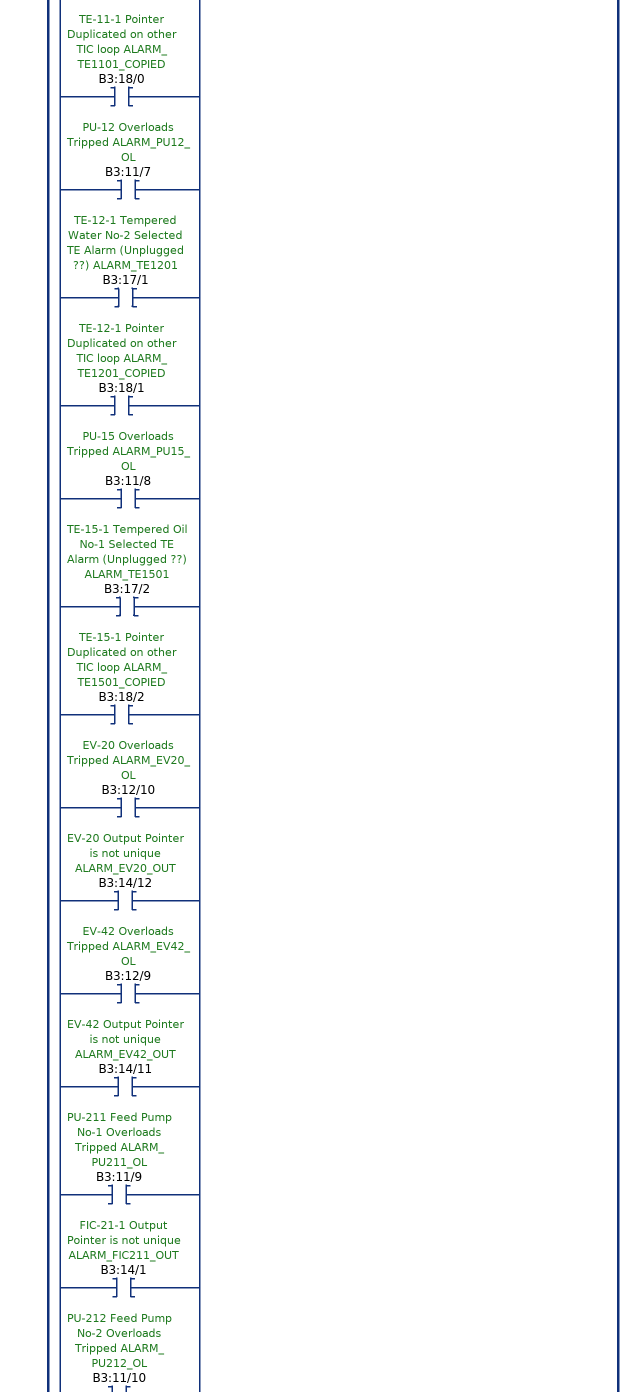

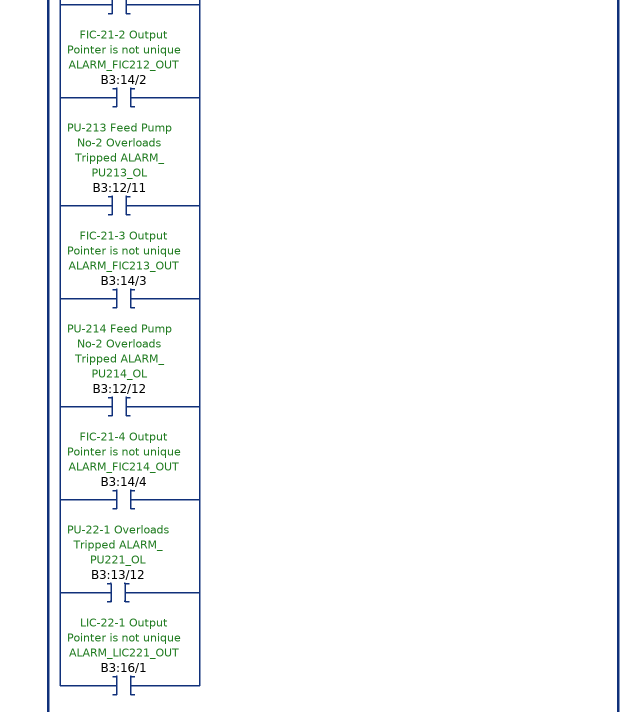
% Rung: 4 %
% This Rung Sets a Bit
% used by the HMI's
% to Determine Whether Alarm Status Page 1
% Has an Active Alarm %
SOR BST XIC B3:12/3 NXB XIC B3:12/0 NXB XIC B3:11/3 NXB XIC B3:14/10 NXB XIC B3:13/13 NXB XIC B3:13/14 NXB XIC B3:11/0 NXB XIC B3:11/1 NXB XIC B3:14/8 NXB XIC B3:11/2 NXB XIC B3:14/9 NXB XIC B3:11/6 NXB XIC B3:17/0 NXB XIC B3:18/0 NXB XIC B3:11/7 NXB XIC B3:17/1 NXB XIC B3:18/1 NXB XIC B3:11/8 NXB XIC B3:17/2 NXB XIC B3:18/2 NXB XIC B3:12/10 NXB XIC B3:14/12 NXB XIC B3:12/9 NXB XIC B3:14/11 NXB XIC B3:11/9 NXB XIC B3:14/1 NXB XIC B3:11/10 NXB XIC B3:14/2 NXB XIC B3:12/11 NXB XIC B3:14/3 NXB XIC B3:12/12 NXB XIC B3:14/4 NXB XIC B3:13/12 NXB XIC B3:16/1 BND OTE B3:10/11 EOR
%   B3:12/3  ALARM_FIRE_ALARM  "WFE Test Center Fire Alarm has be Triggered" %
%   B3:12/0  ALARM_E_STOP  "E-Stop Pushbutton has Been Pressed" %
%   B3:11/3  ALARM_AG04_OL  "AG-4 Overloads Tripped" %
%   B3:14/10  ALARM_AG04_OUT  "AG-4 Output Pointer is not unique" %
%   B3:13/13  ALARM_EF1_OL  "EF-1 Process Area Exhaust Fan Overloads Tripped" %
%   B3:13/14  ALARM_EF2_OL  "EF-2 Utility Room Exhaust Fan Overloads Tripped" %
%   B3:11/0  ALARM_EV01_OL  "EV-1 Overloads Tripped" %
%   B3:11/1  ALARM_EV02_OL  "EV-2 Overloads Tripped" %
%   B3:14/8  ALARM_EV02_OUT  "EV-2 Output Pointer is not unique" %
%   B3:11/2  ALARM_EV03_OL  "EV-3 Overloads Tripped" %
%   B3:14/9  ALARM_EV03_OUT  "EV-3 Output Pointer is not unique" %
%   B3:11/6  ALARM_PU11_OL  "PU-11 Overloads Tripped" %
%   B3:17/0  ALARM_TE1101  "TE-11-1 Tempered Water No-1 Selected TE Alarm (Unplugged ??)" %
%   B3:18/0  ALARM_TE1101_COPIED  "TE-11-1 Pointer Duplicated on other TIC loop" %
%   B3:11/7  ALARM_PU12_OL  "PU-12 Overloads Tripped" %
%   B3:17/1  ALARM_TE1201  "TE-12-1 Tempered Water No-2 Selected TE Alarm (Unplugged ??)" %
%   B3:18/1  ALARM_TE1201_COPIED  "TE-12-1 Pointer Duplicated on other TIC loop" %
%   B3:11/8  ALARM_PU15_OL  "PU-15 Overloads Tripped" %
%   B3:17/2  ALARM_TE1501  "TE-15-1 Tempered Oil No-1 Selected TE Alarm (Unplugged ??)" %
%   B3:18/2  ALARM_TE1501_COPIED  "TE-15-1 Pointer Duplicated on other TIC loop" %
%   B3:12/10  ALARM_EV20_OL  "EV-20 Overloads Tripped" %
%   B3:14/12  ALARM_EV20_OUT  "EV-20 Output Pointer is not unique" %
%   B3:12/9  ALARM_EV42_OL  "EV-42 Overloads Tripped" %
%   B3:14/11  ALARM_EV42_OUT  "EV-42 Output Pointer is not unique" %
%   B3:11/9  ALARM_PU211_OL  "PU-211 Feed Pump No-1 Overloads Tripped" %
%   B3:14/1  ALARM_FIC211_OUT  "FIC-21-1 Output Pointer is not unique" %
%   B3:11/10  ALARM_PU212_OL  "PU-212 Feed Pump No-2 Overloads Tripped" %
%   B3:14/2  ALARM_FIC212_OUT  "FIC-21-2 Output Pointer is not unique" %
%   B3:12/11  ALARM_PU213_OL  "PU-213 Feed Pump No-2 Overloads Tripped" %
%   B3:14/3  ALARM_FIC213_OUT  "FIC-21-3 Output Pointer is not unique" %
%   B3:12/12  ALARM_PU214_OL  "PU-214 Feed Pump No-2 Overloads Tripped" %
%   B3:14/4  ALARM_FIC214_OUT  "FIC-21-4 Output Pointer is not unique" %
%   B3:13/12  ALARM_PU221_OL  "PU-22-1 Overloads Tripped" %
%   B3:16/1  ALARM_LIC221_OUT  "LIC-22-1 Output Pointer is not unique" %
%   B3:10/11  ALARM_ACTIVE_PAGE1  "Alarm Active on HMI Page 1 of 3" %

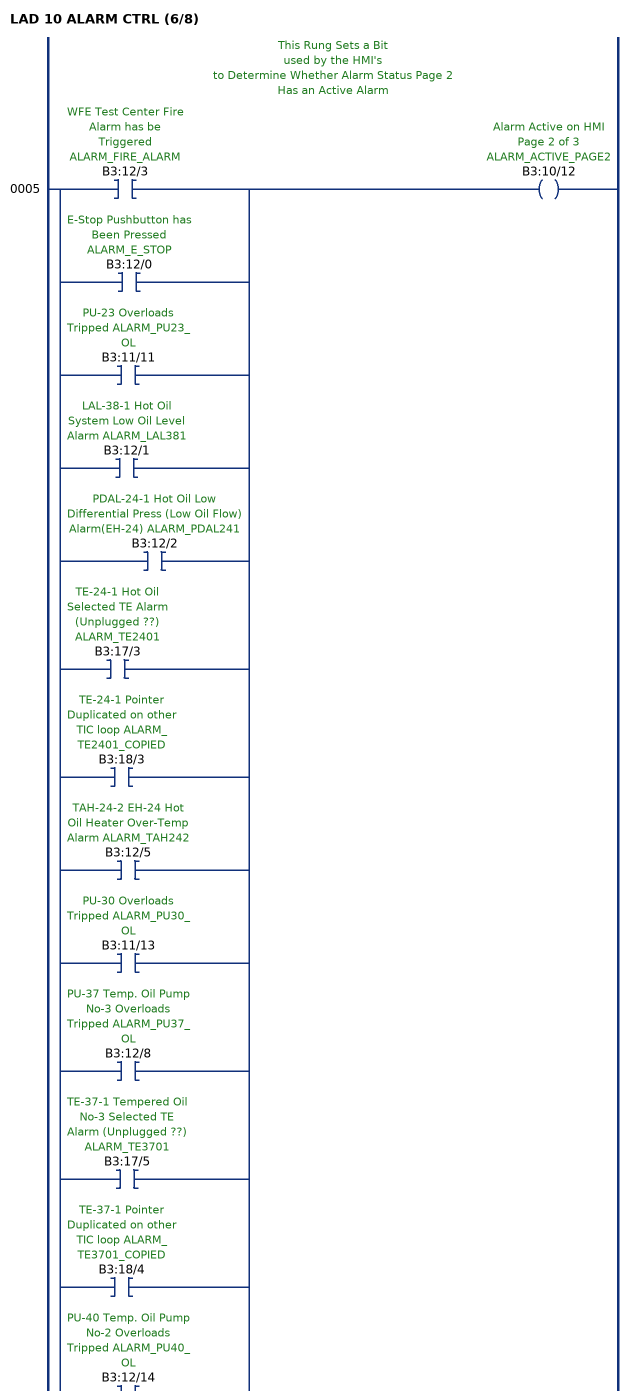

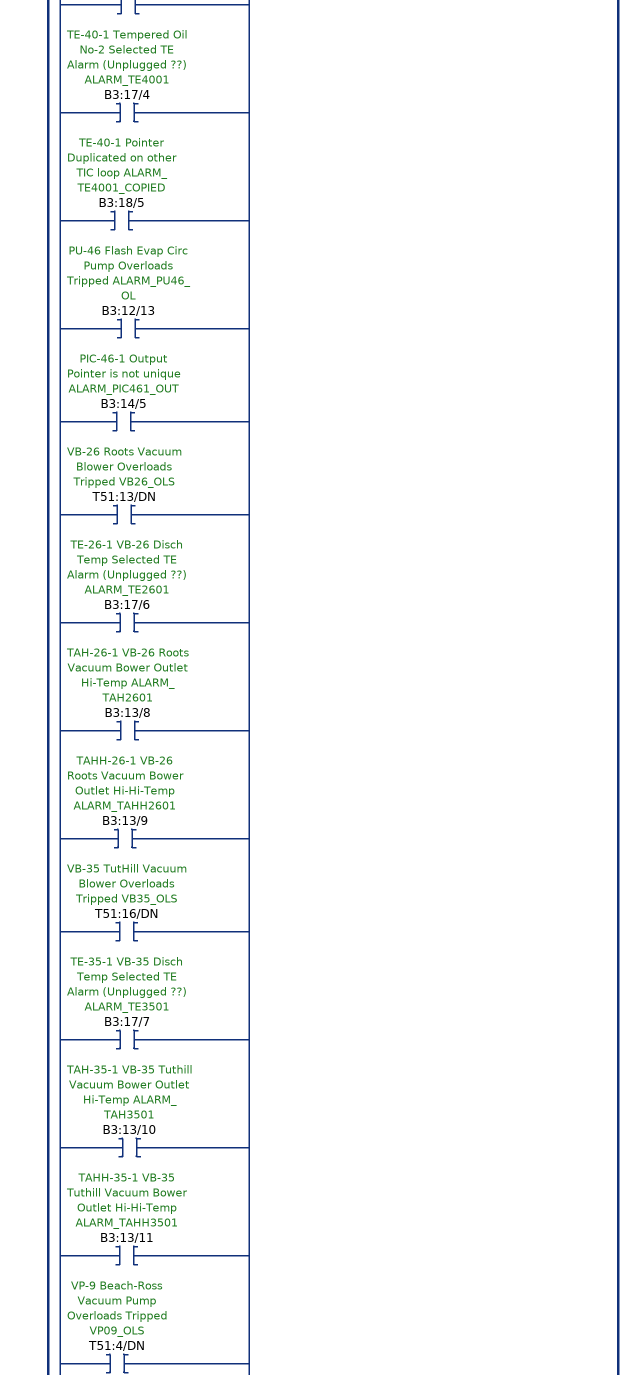

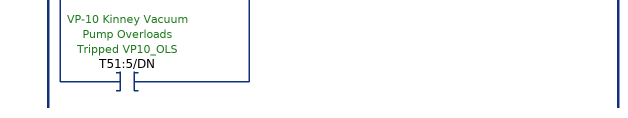
% Rung: 5 %
% This Rung Sets a Bit
% used by the HMI's
% to Determine Whether Alarm Status Page 2
% Has an Active Alarm %
SOR BST XIC B3:12/3 NXB XIC B3:12/0 NXB XIC B3:11/11 NXB XIC B3:12/1 NXB XIC B3:12/2 NXB XIC B3:17/3 NXB XIC B3:18/3 NXB XIC B3:12/5 NXB XIC B3:11/13 NXB XIC B3:12/8 NXB XIC B3:17/5 NXB XIC B3:18/4 NXB XIC B3:12/14 NXB XIC B3:17/4 NXB XIC B3:18/5 NXB XIC B3:12/13 NXB XIC B3:14/5 NXB XIC T51:13/DN NXB XIC B3:17/6 NXB XIC B3:13/8 NXB XIC B3:13/9 NXB XIC T51:16/DN NXB XIC B3:17/7 NXB XIC B3:13/10 NXB XIC B3:13/11 NXB XIC T51:4/DN NXB XIC T51:5/DN BND OTE B3:10/12 EOR
%   B3:12/3  ALARM_FIRE_ALARM  "WFE Test Center Fire Alarm has be Triggered" %
%   B3:12/0  ALARM_E_STOP  "E-Stop Pushbutton has Been Pressed" %
%   B3:11/11  ALARM_PU23_OL  "PU-23 Overloads Tripped" %
%   B3:12/1  ALARM_LAL381  "LAL-38-1 Hot Oil System Low Oil Level Alarm" %
%   B3:12/2  ALARM_PDAL241  "PDAL-24-1 Hot Oil Low Differential Press (Low Oil Flow) Alarm(EH-24)" %
%   B3:17/3  ALARM_TE2401  "TE-24-1 Hot Oil Selected TE Alarm (Unplugged ??)" %
%   B3:18/3  ALARM_TE2401_COPIED  "TE-24-1 Pointer Duplicated on other TIC loop" %
%   B3:12/5  ALARM_TAH242  "TAH-24-2 EH-24 Hot Oil Heater Over-Temp Alarm" %
%   B3:11/13  ALARM_PU30_OL  "PU-30 Overloads Tripped" %
%   B3:12/8  ALARM_PU37_OL  "PU-37 Temp. Oil Pump No-3 Overloads Tripped" %
%   B3:17/5  ALARM_TE3701  "TE-37-1 Tempered Oil No-3 Selected TE Alarm (Unplugged ??)" %
%   B3:18/4  ALARM_TE3701_COPIED  "TE-37-1 Pointer Duplicated on other TIC loop" %
%   B3:12/14  ALARM_PU40_OL  "PU-40 Temp. Oil Pump No-2 Overloads Tripped" %
%   B3:17/4  ALARM_TE4001  "TE-40-1 Tempered Oil No-2 Selected TE Alarm (Unplugged ??)" %
%   B3:18/5  ALARM_TE4001_COPIED  "TE-40-1 Pointer Duplicated on other TIC loop" %
%   B3:12/13  ALARM_PU46_OL  "PU-46 Flash Evap Circ Pump Overloads Tripped" %
%   B3:14/5  ALARM_PIC461_OUT  "PIC-46-1 Output Pointer is not unique" %
%   T51:13/DN  VB26_OLS  "VB-26 Roots Vacuum Blower Overloads Tripped" %
%   B3:17/6  ALARM_TE2601  "TE-26-1 VB-26 Disch Temp Selected TE Alarm (Unplugged ??)" %
%   B3:13/8  ALARM_TAH2601  "TAH-26-1 VB-26 Roots Vacuum Bower Outlet Hi-Temp" %
%   B3:13/9  ALARM_TAHH2601  "TAHH-26-1 VB-26 Roots Vacuum Bower Outlet Hi-Hi-Temp" %
%   T51:16/DN  VB35_OLS  "VB-35 TutHill Vacuum Blower Overloads Tripped" %
%   B3:17/7  ALARM_TE3501  "TE-35-1 VB-35 Disch Temp Selected TE Alarm (Unplugged ??)" %
%   B3:13/10  ALARM_TAH3501  "TAH-35-1 VB-35 Tuthill Vacuum Bower Outlet Hi-Temp" %
%   B3:13/11  ALARM_TAHH3501  "TAHH-35-1 VB-35 Tuthill Vacuum Bower Outlet Hi-Hi-Temp" %
%   T51:4/DN  VP09_OLS  "VP-9 Beach-Ross Vacuum Pump Overloads Tripped" %
%   T51:5/DN  VP10_OLS  "VP-10 Kinney Vacuum Pump Overloads Tripped" %
%   B3:10/12  ALARM_ACTIVE_PAGE2  "Alarm Active on HMI Page 2 of 3" %

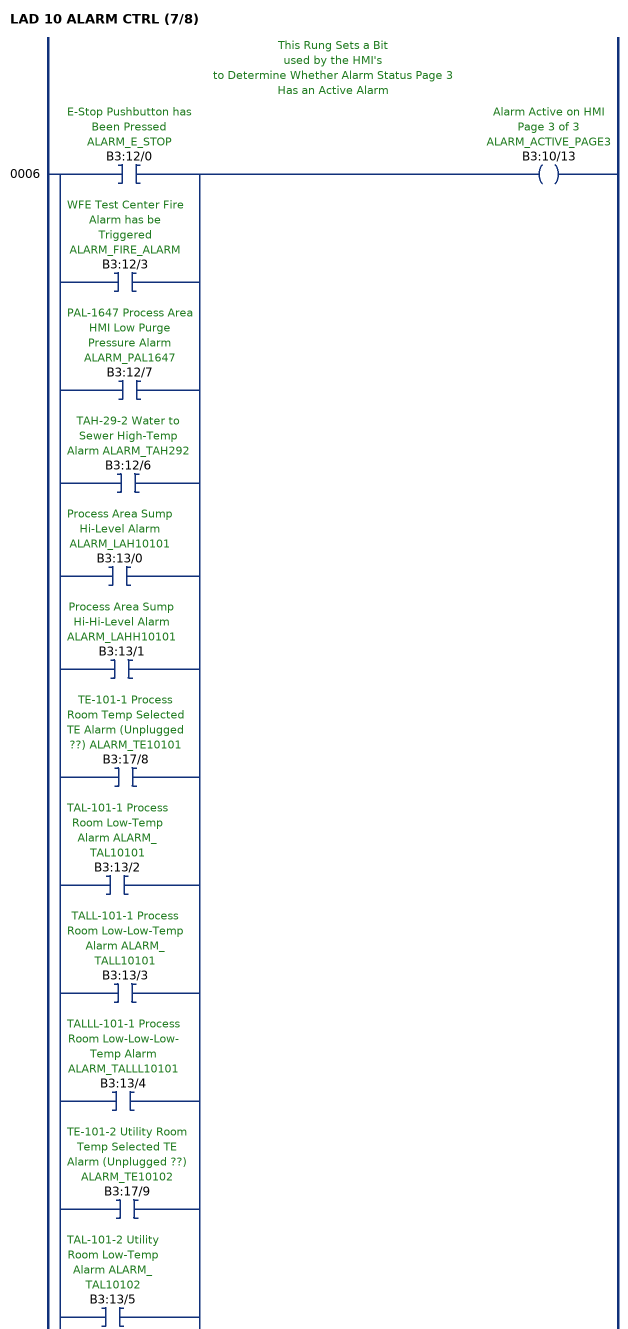

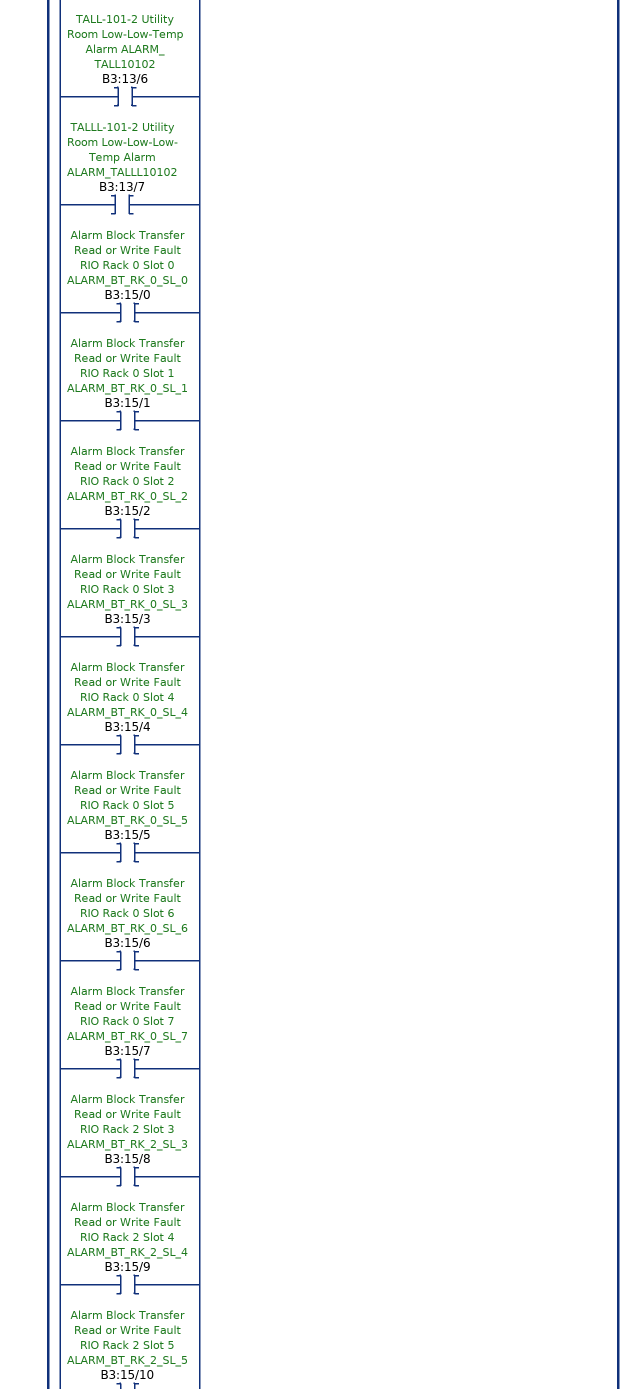

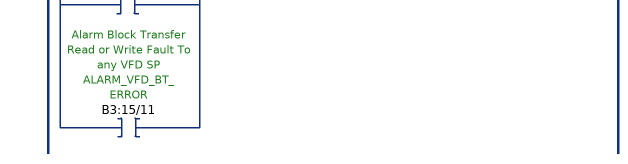
% Rung: 6 %
% This Rung Sets a Bit
% used by the HMI's
% to Determine Whether Alarm Status Page 3
% Has an Active Alarm %
SOR BST XIC B3:12/0 NXB XIC B3:12/3 NXB XIC B3:12/7 NXB XIC B3:12/6 NXB XIC B3:13/0 NXB XIC B3:13/1 NXB XIC B3:17/8 NXB XIC B3:13/2 NXB XIC B3:13/3 NXB XIC B3:13/4 NXB XIC B3:17/9 NXB XIC B3:13/5 NXB XIC B3:13/6 NXB XIC B3:13/7 NXB XIC B3:15/0 NXB XIC B3:15/1 NXB XIC B3:15/2 NXB XIC B3:15/3 NXB XIC B3:15/4 NXB XIC B3:15/5 NXB XIC B3:15/6 NXB XIC B3:15/7 NXB XIC B3:15/8 NXB XIC B3:15/9 NXB XIC B3:15/10 NXB XIC B3:15/11 BND OTE B3:10/13 EOR
%   B3:12/0  ALARM_E_STOP  "E-Stop Pushbutton has Been Pressed" %
%   B3:12/3  ALARM_FIRE_ALARM  "WFE Test Center Fire Alarm has be Triggered" %
%   B3:12/7  ALARM_PAL1647  "PAL-1647 Process Area HMI Low Purge Pressure Alarm" %
%   B3:12/6  ALARM_TAH292  "TAH-29-2 Water to Sewer High-Temp Alarm" %
%   B3:13/0  ALARM_LAH10101  "Process Area Sump Hi-Level Alarm" %
%   B3:13/1  ALARM_LAHH10101  "Process Area Sump Hi-Hi-Level Alarm" %
%   B3:17/8  ALARM_TE10101  "TE-101-1 Process Room Temp Selected TE Alarm (Unplugged ??)" %
%   B3:13/2  ALARM_TAL10101  "TAL-101-1 Process Room Low-Temp Alarm" %
%   B3:13/3  ALARM_TALL10101  "TALL-101-1 Process Room Low-Low-Temp Alarm" %
%   B3:13/4  ALARM_TALLL10101  "TALLL-101-1 Process Room Low-Low-Low-Temp Alarm" %
%   B3:17/9  ALARM_TE10102  "TE-101-2 Utility Room Temp Selected TE Alarm (Unplugged ??)" %
%   B3:13/5  ALARM_TAL10102  "TAL-101-2 Utility Room Low-Temp Alarm" %
%   B3:13/6  ALARM_TALL10102  "TALL-101-2 Utility Room Low-Low-Temp Alarm" %
%   B3:13/7  ALARM_TALLL10102  "TALLL-101-2 Utility Room Low-Low-Low-Temp Alarm" %
%   B3:15/0  ALARM_BT_RK_0_SL_0  "Alarm Block Transfer Read or Write Fault RIO Rack 0 Slot 0" %
%   B3:15/1  ALARM_BT_RK_0_SL_1  "Alarm Block Transfer Read or Write Fault RIO Rack 0 Slot 1" %
%   B3:15/2  ALARM_BT_RK_0_SL_2  "Alarm Block Transfer Read or Write Fault RIO Rack 0 Slot 2" %
%   B3:15/3  ALARM_BT_RK_0_SL_3  "Alarm Block Transfer Read or Write Fault RIO Rack 0 Slot 3" %
%   B3:15/4  ALARM_BT_RK_0_SL_4  "Alarm Block Transfer Read or Write Fault RIO Rack 0 Slot 4" %
%   B3:15/5  ALARM_BT_RK_0_SL_5  "Alarm Block Transfer Read or Write Fault RIO Rack 0 Slot 5" %
%   B3:15/6  ALARM_BT_RK_0_SL_6  "Alarm Block Transfer Read or Write Fault RIO Rack 0 Slot 6" %
%   B3:15/7  ALARM_BT_RK_0_SL_7  "Alarm Block Transfer Read or Write Fault RIO Rack 0 Slot 7" %
%   B3:15/8  ALARM_BT_RK_2_SL_3  "Alarm Block Transfer Read or Write Fault RIO Rack 2 Slot 3" %
%   B3:15/9  ALARM_BT_RK_2_SL_4  "Alarm Block Transfer Read or Write Fault RIO Rack 2 Slot 4" %
%   B3:15/10  ALARM_BT_RK_2_SL_5  "Alarm Block Transfer Read or Write Fault RIO Rack 2 Slot 5" %
%   B3:15/11  ALARM_VFD_BT_ERROR  "Alarm Block Transfer Read or Write Fault To any VFD SP" %
%   B3:10/13  ALARM_ACTIVE_PAGE3  "Alarm Active on HMI Page 3 of 3" %

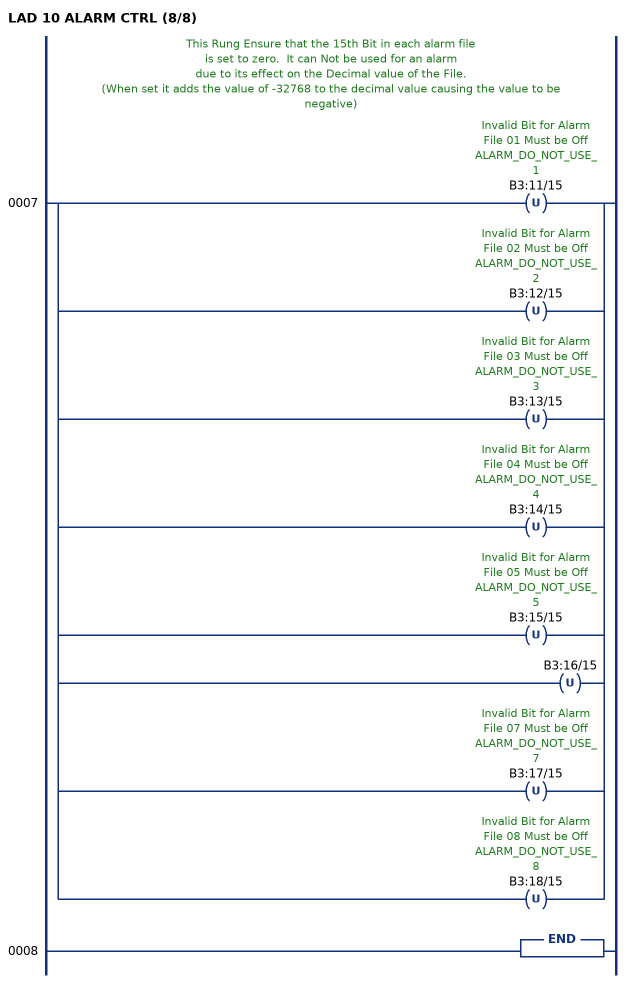
% Rung: 7 %
% This Rung Ensure that the 15th Bit in each alarm file
% is set to zero.  It can Not be used for an alarm
% due to its effect on the Decimal value of the File.
% (When set it adds the value of -32768 to the decimal value causing the value to be negative) %
SOR BST OTU B3:11/15 NXB OTU B3:12/15 NXB OTU B3:13/15 NXB OTU B3:14/15 NXB OTU B3:15/15 NXB OTU B3:16/15 NXB OTU B3:17/15 NXB OTU B3:18/15 BND EOR
%   B3:11/15  ALARM_DO_NOT_USE_1  "Invalid Bit for Alarm File 01 Must be Off" %
%   B3:12/15  ALARM_DO_NOT_USE_2  "Invalid Bit for Alarm File 02 Must be Off" %
%   B3:13/15  ALARM_DO_NOT_USE_3  "Invalid Bit for Alarm File 03 Must be Off" %
%   B3:14/15  ALARM_DO_NOT_USE_4  "Invalid Bit for Alarm File 04 Must be Off" %
%   B3:15/15  ALARM_DO_NOT_USE_5  "Invalid Bit for Alarm File 05 Must be Off" %
%   B3:17/15  ALARM_DO_NOT_USE_7  "Invalid Bit for Alarm File 07 Must be Off" %
%   B3:18/15  ALARM_DO_NOT_USE_8  "Invalid Bit for Alarm File 08 Must be Off" %
% Rung: 8 %
SOR END EOR

LADDER 11 "ALARMS"    % Process Alarms %
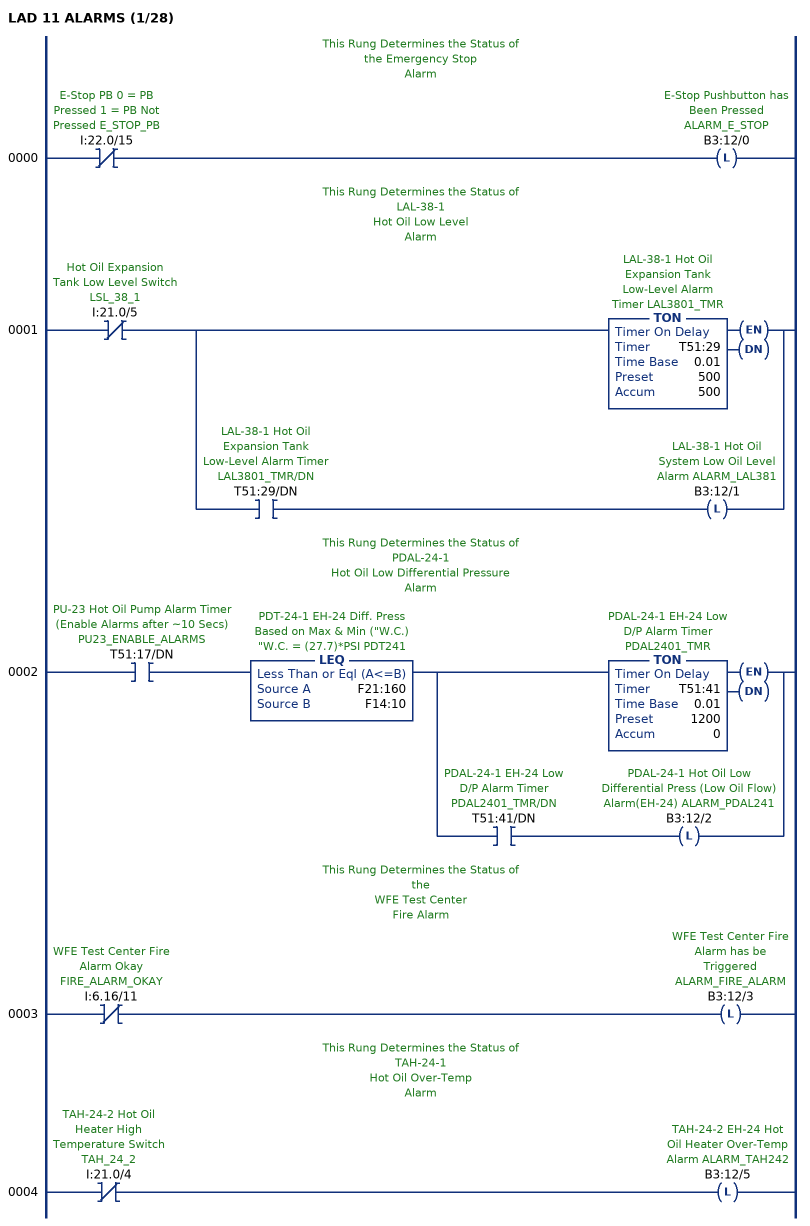
% Rung: 0 %
% This Rung Determines the Status of
% the Emergency Stop
% Alarm %
SOR XIO I:22.0/15 OTL B3:12/0 EOR
%   I:22.0/15  E_STOP_PB  "E-Stop PB 0 = PB Pressed 1 = PB Not Pressed" %
%   B3:12/0  ALARM_E_STOP  "E-Stop Pushbutton has Been Pressed" %
% Rung: 1 %
% This Rung Determines the Status of
% LAL-38-1
% Hot Oil Low Level
% Alarm %
SOR XIO I:21.0/5 BST TON T51:29 0.01 500 500 NXB XIC T51:29/DN OTL B3:12/1 BND EOR
%   I:21.0/5  LSL_38_1  "Hot Oil Expansion Tank Low Level Switch" %
%   T51:29  LAL3801_TMR  "LAL-38-1 Hot Oil Expansion Tank Low-Level Alarm Timer" %
%   B3:12/1  ALARM_LAL381  "LAL-38-1 Hot Oil System Low Oil Level Alarm" %
% Rung: 2 %
% This Rung Determines the Status of
% PDAL-24-1
% Hot Oil Low Differential Pressure
% Alarm %
SOR XIC T51:17/DN LEQ F21:160 F14:10 BST TON T51:41 0.01 1200 0 NXB XIC T51:41/DN OTL B3:12/2 BND EOR
%   T51:17/DN  PU23_ENABLE_ALARMS  "PU-23 Hot Oil Pump Alarm Timer (Enable Alarms after ~10 Secs)" %
%   F21:160  PDT241  "PDT-24-1 EH-24 Diff. Press Based on Max & Min ("W.C.) "W.C. = (27.7)*PSI" %
%   F14:10  PDAL2401_SP  "PDAL-24-1 Hot Oil Low Differential Press (Low Oil Flow) SP" %
%   T51:41  PDAL2401_TMR  "PDAL-24-1 EH-24 Low D/P Alarm Timer" %
%   B3:12/2  ALARM_PDAL241  "PDAL-24-1 Hot Oil Low Differential Press (Low Oil Flow) Alarm(EH-24)" %
% Rung: 3 %
% This Rung Determines the Status of
% the
% WFE Test Center
% Fire Alarm %
SOR XIO I:6.16/11 OTL B3:12/3 EOR
%   I:6.16/11  FIRE_ALARM_OKAY  "WFE Test Center Fire Alarm Okay" %
%   B3:12/3  ALARM_FIRE_ALARM  "WFE Test Center Fire Alarm has be Triggered" %
% Rung: 4 %
% This Rung Determines the Status of
% TAH-24-1
% Hot Oil Over-Temp
% Alarm %
SOR XIO I:21.0/4 OTL B3:12/5 EOR
%   I:21.0/4  TAH_24_2  "TAH-24-2 Hot Oil Heater High Temperature Switch" %
%   B3:12/5  ALARM_TAH242  "TAH-24-2 EH-24 Hot Oil Heater Over-Temp Alarm" %

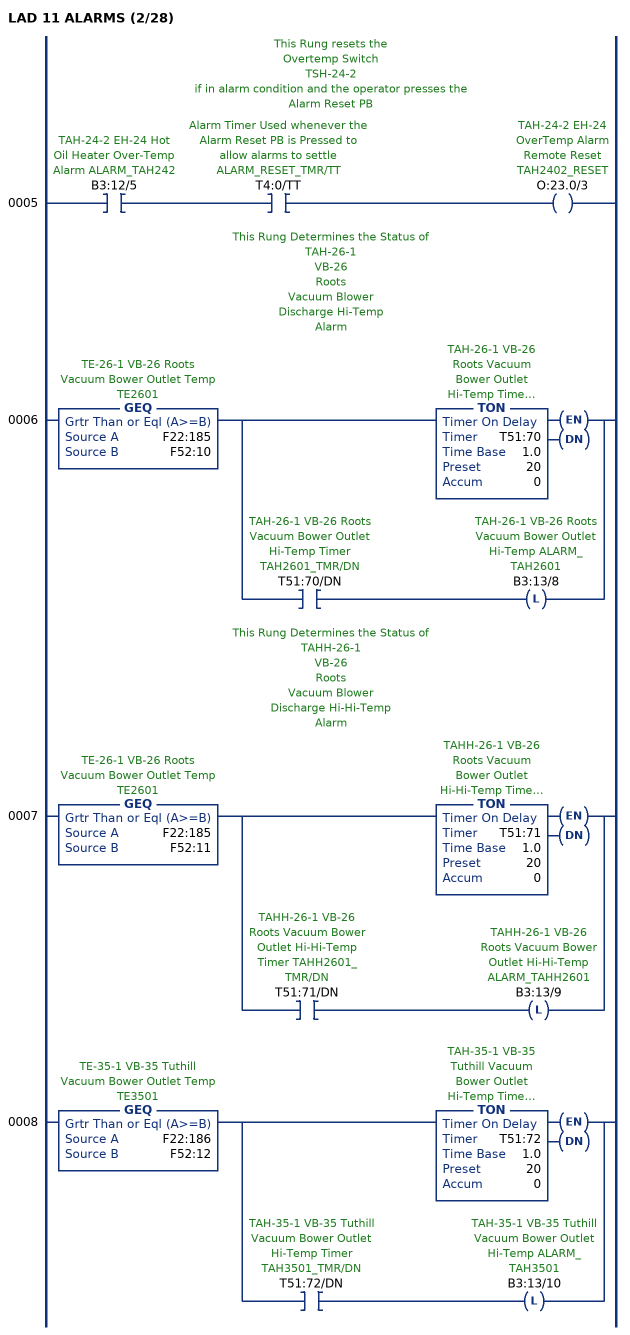
% Rung: 5 %
% This Rung resets the
% Overtemp Switch
% TSH-24-2
% if in alarm condition and the operator presses the
% Alarm Reset PB %
SOR XIC B3:12/5 XIC T4:0/TT OTE O:23.0/3 EOR
%   B3:12/5  ALARM_TAH242  "TAH-24-2 EH-24 Hot Oil Heater Over-Temp Alarm" %
%   T4:0  ALARM_RESET_TMR  "Alarm Timer Used whenever the Alarm Reset PB is Pressed to allow alarms to settle" %
%   O:23.0/3  TAH2402_RESET  "TAH-24-2 EH-24 OverTemp Alarm Remote Reset" %
% Rung: 6 %
% This Rung Determines the Status of
% TAH-26-1
% VB-26
% Roots
% Vacuum Blower
% Discharge Hi-Temp
% Alarm %
SOR GEQ F22:185 F52:10 BST TON T51:70 1.0 20 0 NXB XIC T51:70/DN OTL B3:13/8 BND EOR
%   F22:185  TE2601  "TE-26-1 VB-26 Roots Vacuum Bower Outlet Temp" %
%   F52:10  TAH2601_SP  "TAH-26-1 VB-26 Roots Blower Hi-Temp Alarm Setpoint" %
%   T51:70  TAH2601_TMR  "TAH-26-1 VB-26 Roots Vacuum Bower Outlet Hi-Temp Timer" %
%   B3:13/8  ALARM_TAH2601  "TAH-26-1 VB-26 Roots Vacuum Bower Outlet Hi-Temp" %
% Rung: 7 %
% This Rung Determines the Status of
% TAHH-26-1
% VB-26
% Roots
% Vacuum Blower
% Discharge Hi-Hi-Temp
% Alarm %
SOR GEQ F22:185 F52:11 BST TON T51:71 1.0 20 0 NXB XIC T51:71/DN OTL B3:13/9 BND EOR
%   F22:185  TE2601  "TE-26-1 VB-26 Roots Vacuum Bower Outlet Temp" %
%   F52:11  TAHH2601_SP  "TAHH-26-1 VB-26 Roots Blower Hi-Hi-Temp Alarm Setpoint" %
%   T51:71  TAHH2601_TMR  "TAHH-26-1 VB-26 Roots Vacuum Bower Outlet Hi-Hi-Temp Timer" %
%   B3:13/9  ALARM_TAHH2601  "TAHH-26-1 VB-26 Roots Vacuum Bower Outlet Hi-Hi-Temp" %
% Rung: 8 %
SOR GEQ F22:186 F52:12 BST TON T51:72 1.0 20 0 NXB XIC T51:72/DN OTL B3:13/10 BND EOR
%   F22:186  TE3501  "TE-35-1 VB-35 Tuthill Vacuum Bower Outlet Temp" %
%   F52:12  TAH3501_SP  "TAH-35-1 VB-35 Tuthill Blower Hi-Temp Alarm Setpoint" %
%   T51:72  TAH3501_TMR  "TAH-35-1 VB-35 Tuthill Vacuum Bower Outlet Hi-Temp Timer" %
%   B3:13/10  ALARM_TAH3501  "TAH-35-1 VB-35 Tuthill Vacuum Bower Outlet Hi-Temp" %

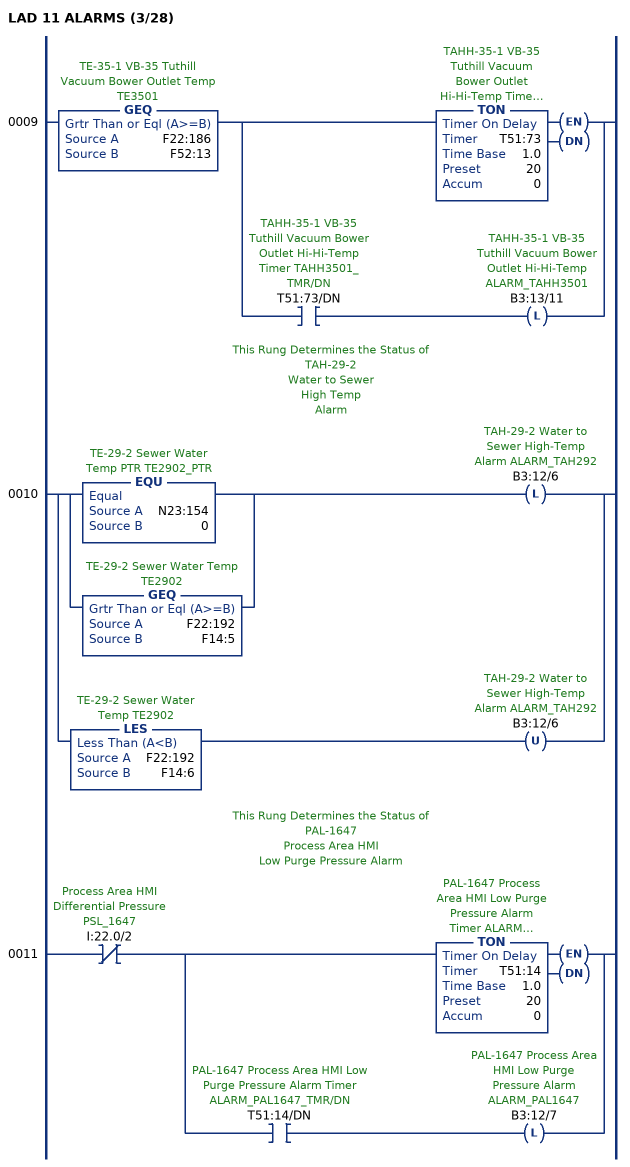
% Rung: 9 %
SOR GEQ F22:186 F52:13 BST TON T51:73 1.0 20 0 NXB XIC T51:73/DN OTL B3:13/11 BND EOR
%   F22:186  TE3501  "TE-35-1 VB-35 Tuthill Vacuum Bower Outlet Temp" %
%   F52:13  TAHH3501_SP  "TAH-35-1 VB-35 Tuthill Blower Hi-Hi-Temp Alarm Setpoint" %
%   T51:73  TAHH3501_TMR  "TAHH-35-1 VB-35 Tuthill Vacuum Bower Outlet Hi-Hi-Temp Timer" %
%   B3:13/11  ALARM_TAHH3501  "TAHH-35-1 VB-35 Tuthill Vacuum Bower Outlet Hi-Hi-Temp" %
% Rung: 10 %
% This Rung Determines the Status of
% TAH-29-2
% Water to Sewer
% High Temp
% Alarm %
SOR BST BST EQU N23:154 0 NXB GEQ F22:192 F14:5 BND OTL B3:12/6 NXB LES F22:192 F14:6 OTU B3:12/6 BND EOR
%   N23:154  TE2902_PTR  "TE-29-2 Sewer Water Temp PTR" %
%   F22:192  TE2902  "TE-29-2 Sewer Water Temp" %
%   F14:5  TAH2902_SP  "TAH-29-2 Water to Sewer HIGH Temp Alarm Setpoint" %
%   B3:12/6  ALARM_TAH292  "TAH-29-2 Water to Sewer High-Temp Alarm" %
%   F14:6  TAH2902_RESET_SP  "TAH-29-2 Water to Sewer HIGH Temp Alarm Clear Setpoint" %
% Rung: 11 %
% This Rung Determines the Status of
% PAL-1647
% Process Area HMI
% Low Purge Pressure Alarm %
SOR XIO I:22.0/2 BST TON T51:14 1.0 20 0 NXB XIC T51:14/DN OTL B3:12/7 BND EOR
%   I:22.0/2  PSL_1647  "Process Area HMI Differential Pressure" %
%   T51:14  ALARM_PAL1647_TMR  "PAL-1647 Process Area HMI Low Purge Pressure Alarm Timer" %
%   B3:12/7  ALARM_PAL1647  "PAL-1647 Process Area HMI Low Purge Pressure Alarm" %

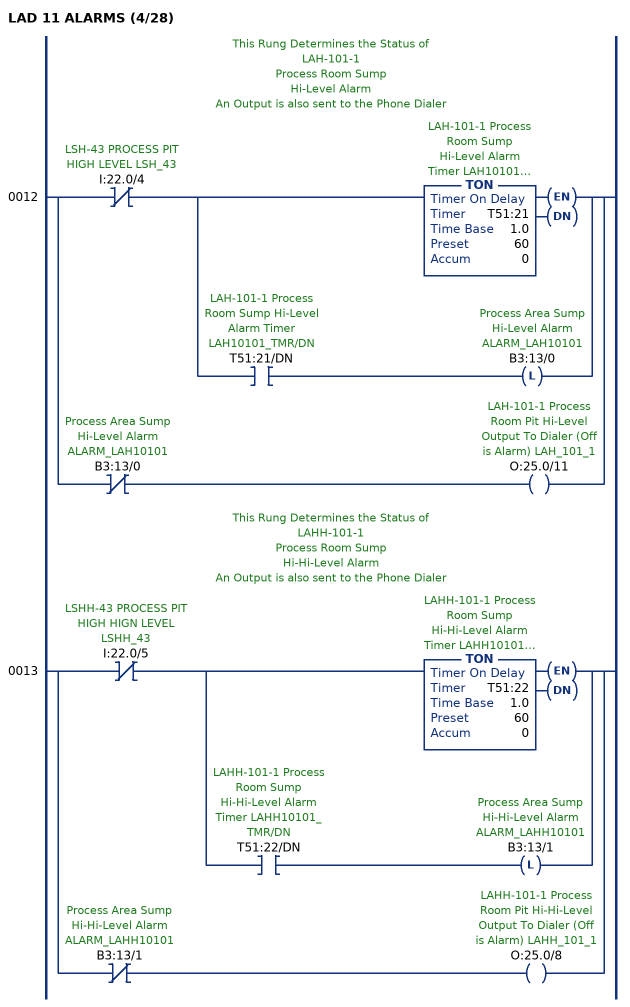
% Rung: 12 %
% This Rung Determines the Status of
% LAH-101-1
% Process Room Sump
% Hi-Level Alarm
% An Output is also sent to the Phone Dialer %
SOR BST XIO I:22.0/4 BST TON T51:21 1.0 60 0 NXB XIC T51:21/DN OTL B3:13/0 BND NXB XIO B3:13/0 OTE O:25.0/11 BND EOR
%   I:22.0/4  LSH_43  "LSH-43 PROCESS PIT HIGH LEVEL" %
%   T51:21  LAH10101_TMR  "LAH-101-1 Process Room Sump Hi-Level Alarm Timer" %
%   B3:13/0  ALARM_LAH10101  "Process Area Sump Hi-Level Alarm" %
%   O:25.0/11  LAH_101_1  "LAH-101-1 Process Room Pit Hi-Level Output To Dialer (Off is Alarm)" %
% Rung: 13 %
% This Rung Determines the Status of
% LAHH-101-1
% Process Room Sump
% Hi-Hi-Level Alarm
% An Output is also sent to the Phone Dialer %
SOR BST XIO I:22.0/5 BST TON T51:22 1.0 60 0 NXB XIC T51:22/DN OTL B3:13/1 BND NXB XIO B3:13/1 OTE O:25.0/8 BND EOR
%   I:22.0/5  LSHH_43  "LSHH-43 PROCESS PIT HIGH HIGN LEVEL" %
%   T51:22  LAHH10101_TMR  "LAHH-101-1 Process Room Sump Hi-Hi-Level Alarm Timer" %
%   B3:13/1  ALARM_LAHH10101  "Process Area Sump Hi-Hi-Level Alarm" %
%   O:25.0/8  LAHH_101_1  "LAHH-101-1 Process Room Pit Hi-Hi-Level Output To Dialer (Off is Alarm)" %

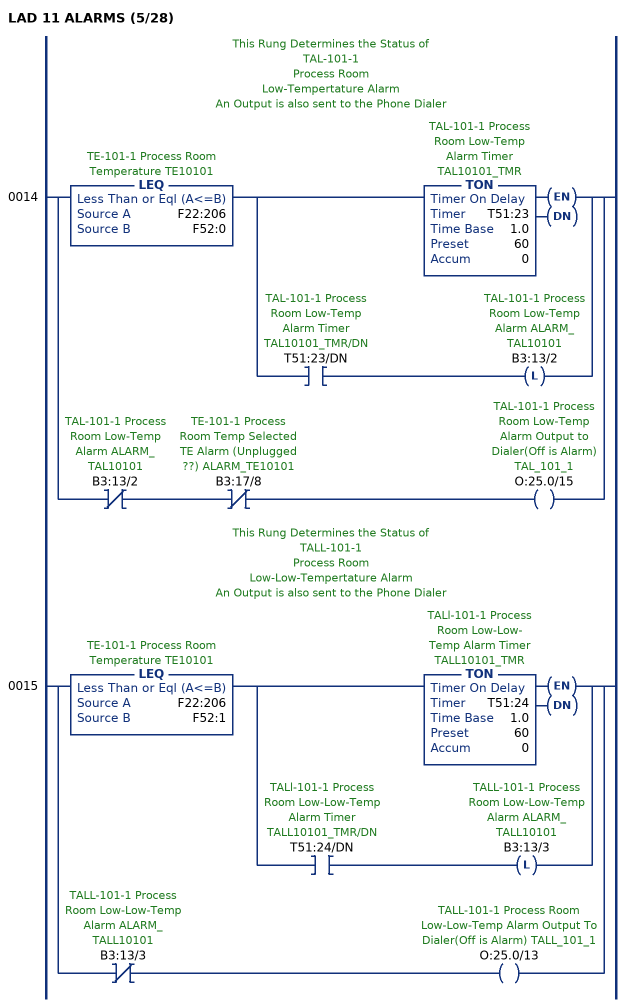
% Rung: 14 %
% This Rung Determines the Status of
% TAL-101-1
% Process Room
% Low-Tempertature Alarm
% An Output is also sent to the Phone Dialer %
SOR BST LEQ F22:206 F52:0 BST TON T51:23 1.0 60 0 NXB XIC T51:23/DN OTL B3:13/2 BND NXB XIO B3:13/2 XIO B3:17/8 OTE O:25.0/15 BND EOR
%   F22:206  TE10101  "TE-101-1 Process Room Temperature" %
%   F52:0  TAL10101_SP  "TAL-101-1 Process Room Low-Temp Alarm Setpoint" %
%   T51:23  TAL10101_TMR  "TAL-101-1 Process Room Low-Temp Alarm Timer" %
%   B3:13/2  ALARM_TAL10101  "TAL-101-1 Process Room Low-Temp Alarm" %
%   B3:17/8  ALARM_TE10101  "TE-101-1 Process Room Temp Selected TE Alarm (Unplugged ??)" %
%   O:25.0/15  TAL_101_1  "TAL-101-1 Process Room Low-Temp Alarm Output to Dialer(Off is Alarm)" %
% Rung: 15 %
% This Rung Determines the Status of
% TALL-101-1
% Process Room
% Low-Low-Tempertature Alarm
% An Output is also sent to the Phone Dialer %
SOR BST LEQ F22:206 F52:1 BST TON T51:24 1.0 60 0 NXB XIC T51:24/DN OTL B3:13/3 BND NXB XIO B3:13/3 OTE O:25.0/13 BND EOR
%   F22:206  TE10101  "TE-101-1 Process Room Temperature" %
%   F52:1  TALL10101_SP  "TALL-101-1 Process Room Low-Low-Temp Alarm Setpoint" %
%   T51:24  TALL10101_TMR  "TALl-101-1 Process Room Low-Low-Temp Alarm Timer" %
%   B3:13/3  ALARM_TALL10101  "TALL-101-1 Process Room Low-Low-Temp Alarm" %
%   O:25.0/13  TALL_101_1  "TALL-101-1 Process Room Low-Low-Temp Alarm Output To Dialer(Off is Alarm)" %

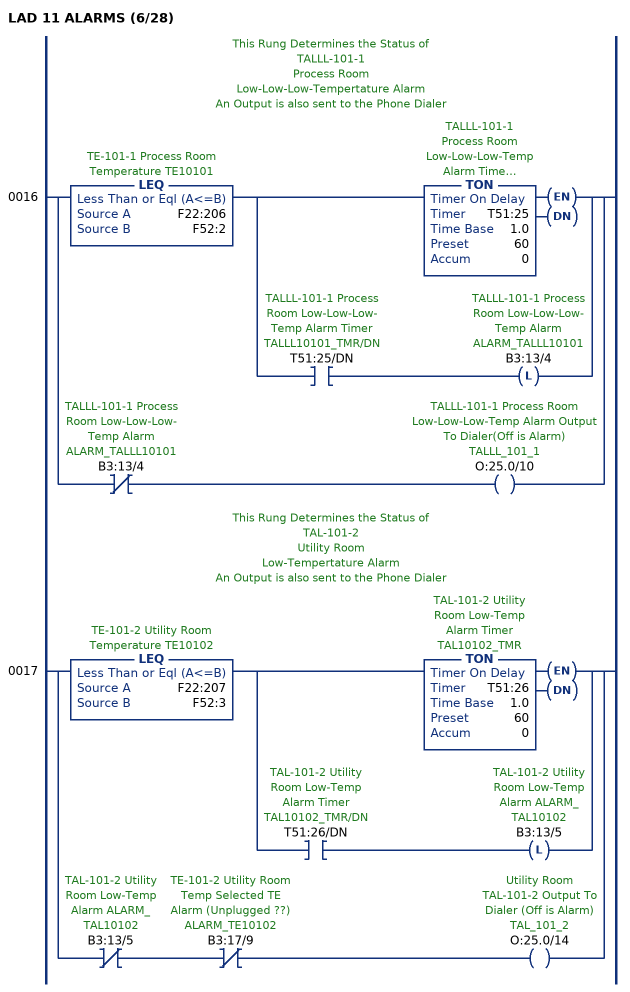
% Rung: 16 %
% This Rung Determines the Status of
% TALLL-101-1
% Process Room
% Low-Low-Low-Tempertature Alarm
% An Output is also sent to the Phone Dialer %
SOR BST LEQ F22:206 F52:2 BST TON T51:25 1.0 60 0 NXB XIC T51:25/DN OTL B3:13/4 BND NXB XIO B3:13/4 OTE O:25.0/10 BND EOR
%   F22:206  TE10101  "TE-101-1 Process Room Temperature" %
%   F52:2  TALLL10101_SP  "TALLL-101-1 Process Room Low-Low-Low-Temp Alarm Setpoint" %
%   T51:25  TALLL10101_TMR  "TALLL-101-1 Process Room Low-Low-Low-Temp Alarm Timer" %
%   B3:13/4  ALARM_TALLL10101  "TALLL-101-1 Process Room Low-Low-Low-Temp Alarm" %
%   O:25.0/10  TALLL_101_1  "TALLL-101-1 Process Room Low-Low-Low-Temp Alarm Output To Dialer(Off is Alarm)" %
% Rung: 17 %
% This Rung Determines the Status of
% TAL-101-2
% Utility Room
% Low-Tempertature Alarm
% An Output is also sent to the Phone Dialer %
SOR BST LEQ F22:207 F52:3 BST TON T51:26 1.0 60 0 NXB XIC T51:26/DN OTL B3:13/5 BND NXB XIO B3:13/5 XIO B3:17/9 OTE O:25.0/14 BND EOR
%   F22:207  TE10102  "TE-101-2 Utility Room Temperature" %
%   F52:3  TAL10102_SP  "TAL-101-2 Utility Room Low-Temp Alarm Setpoint" %
%   T51:26  TAL10102_TMR  "TAL-101-2 Utility Room Low-Temp Alarm Timer" %
%   B3:13/5  ALARM_TAL10102  "TAL-101-2 Utility Room Low-Temp Alarm" %
%   B3:17/9  ALARM_TE10102  "TE-101-2 Utility Room Temp Selected TE Alarm (Unplugged ??)" %
%   O:25.0/14  TAL_101_2  "Utility Room TAL-101-2 Output To Dialer (Off is Alarm)" %

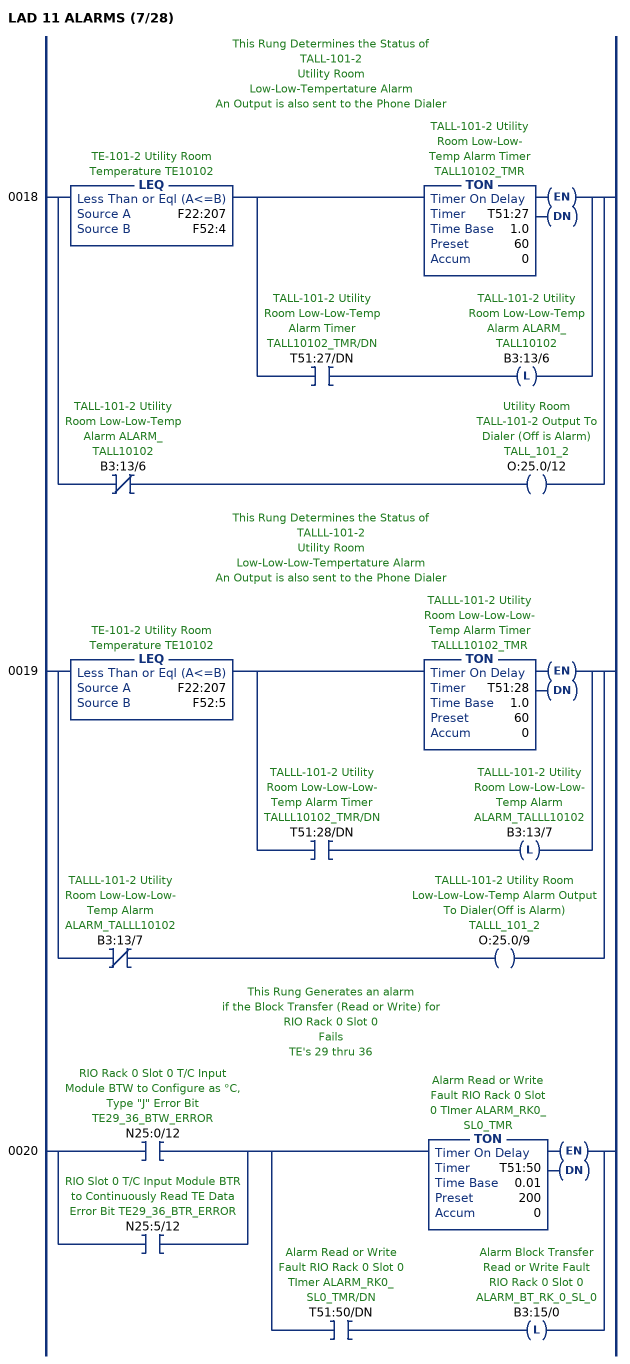
% Rung: 18 %
% This Rung Determines the Status of
% TALL-101-2
% Utility Room
% Low-Low-Tempertature Alarm
% An Output is also sent to the Phone Dialer %
SOR BST LEQ F22:207 F52:4 BST TON T51:27 1.0 60 0 NXB XIC T51:27/DN OTL B3:13/6 BND NXB XIO B3:13/6 OTE O:25.0/12 BND EOR
%   F22:207  TE10102  "TE-101-2 Utility Room Temperature" %
%   F52:4  TALL10102_SP  "TALL-101-2 Utility Room Low-Low-Temp Alarm Setpoint" %
%   T51:27  TALL10102_TMR  "TALL-101-2 Utility Room Low-Low-Temp Alarm Timer" %
%   B3:13/6  ALARM_TALL10102  "TALL-101-2 Utility Room Low-Low-Temp Alarm" %
%   O:25.0/12  TALL_101_2  "Utility Room TALL-101-2 Output To Dialer (Off is Alarm)" %
% Rung: 19 %
% This Rung Determines the Status of
% TALLL-101-2
% Utility Room
% Low-Low-Low-Tempertature Alarm
% An Output is also sent to the Phone Dialer %
SOR BST LEQ F22:207 F52:5 BST TON T51:28 1.0 60 0 NXB XIC T51:28/DN OTL B3:13/7 BND NXB XIO B3:13/7 OTE O:25.0/9 BND EOR
%   F22:207  TE10102  "TE-101-2 Utility Room Temperature" %
%   F52:5  TALLL10102_SP  "TALLL-101-2 Utility Room Low-Low-Low-Temp Alarm Setpoint" %
%   T51:28  TALLL10102_TMR  "TALLL-101-2 Utility Room Low-Low-Low-Temp Alarm Timer" %
%   B3:13/7  ALARM_TALLL10102  "TALLL-101-2 Utility Room Low-Low-Low-Temp Alarm" %
%   O:25.0/9  TALLL_101_2  "TALLL-101-2 Utility Room Low-Low-Low-Temp Alarm Output To Dialer(Off is Alarm)" %
% Rung: 20 %
% This Rung Generates an alarm
% if the Block Transfer (Read or Write) for
% RIO Rack 0 Slot 0
% Fails
% TE's 29 thru 36 %
SOR BST XIC N25:0/12 NXB XIC N25:5/12 BND BST TON T51:50 0.01 200 0 NXB XIC T51:50/DN OTL B3:15/0 BND EOR
%   N25:0/12  TE29_36_BTW_ERROR  "RIO Rack 0 Slot 0 T/C Input Module BTW to Configure as °C, Type "J" Error Bit" %
%   N25:5/12  TE29_36_BTR_ERROR  "RIO Slot 0 T/C Input Module BTR to Continuously Read TE Data Error Bit" %
%   T51:50  ALARM_RK0_SL0_TMR  "Alarm Read or Write Fault RIO Rack 0 Slot 0 TImer" %
%   B3:15/0  ALARM_BT_RK_0_SL_0  "Alarm Block Transfer Read or Write Fault RIO Rack 0 Slot 0" %

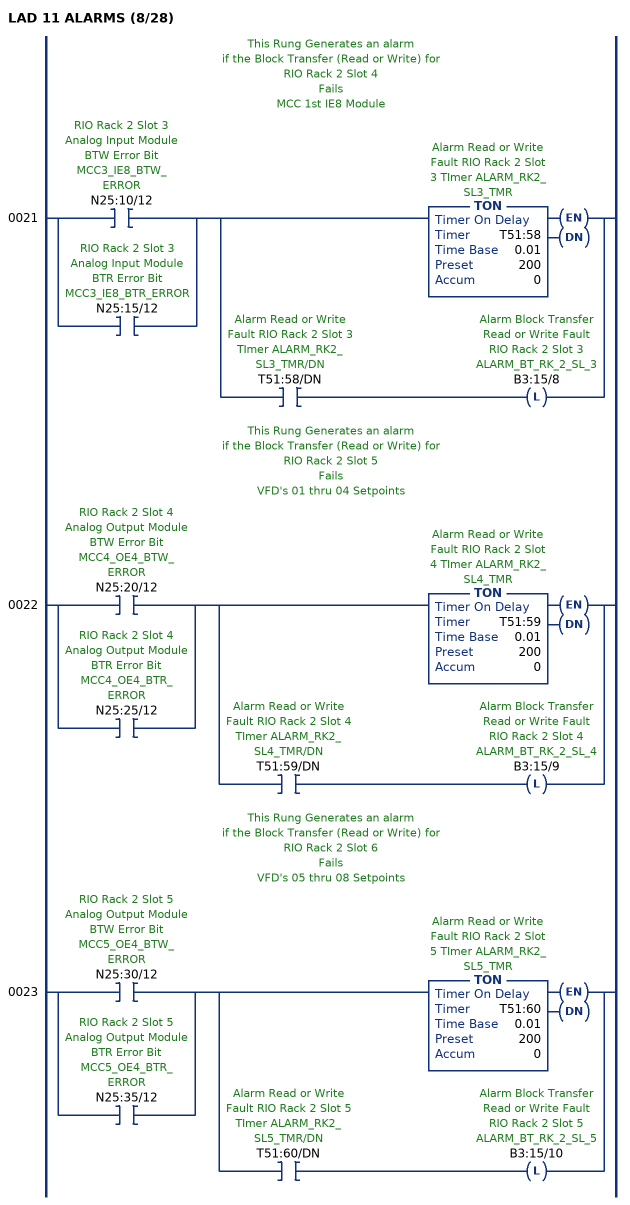
% Rung: 21 %
% This Rung Generates an alarm
% if the Block Transfer (Read or Write) for
% RIO Rack 2 Slot 4
% Fails
%   MCC 1st IE8 Module %
SOR BST XIC N25:10/12 NXB XIC N25:15/12 BND BST TON T51:58 0.01 200 0 NXB XIC T51:58/DN OTL B3:15/8 BND EOR
%   N25:10/12  MCC3_IE8_BTW_ERROR  "RIO Rack 2 Slot 3 Analog Input Module BTW Error Bit" %
%   N25:15/12  MCC3_IE8_BTR_ERROR  "RIO Rack 2 Slot 3 Analog Input Module BTR Error Bit" %
%   T51:58  ALARM_RK2_SL3_TMR  "Alarm Read or Write Fault RIO Rack 2 Slot 3 TImer" %
%   B3:15/8  ALARM_BT_RK_2_SL_3  "Alarm Block Transfer Read or Write Fault RIO Rack 2 Slot 3" %
% Rung: 22 %
% This Rung Generates an alarm
% if the Block Transfer (Read or Write) for
% RIO Rack 2 Slot 5
% Fails
% VFD's 01 thru 04 Setpoints %
SOR BST XIC N25:20/12 NXB XIC N25:25/12 BND BST TON T51:59 0.01 200 0 NXB XIC T51:59/DN OTL B3:15/9 BND EOR
%   N25:20/12  MCC4_OE4_BTW_ERROR  "RIO Rack 2 Slot 4 Analog Output Module BTW Error Bit" %
%   N25:25/12  MCC4_OE4_BTR_ERROR  "RIO Rack 2 Slot 4 Analog Output Module BTR Error Bit" %
%   T51:59  ALARM_RK2_SL4_TMR  "Alarm Read or Write Fault RIO Rack 2 Slot 4 TImer" %
%   B3:15/9  ALARM_BT_RK_2_SL_4  "Alarm Block Transfer Read or Write Fault RIO Rack 2 Slot 4" %
% Rung: 23 %
% This Rung Generates an alarm
% if the Block Transfer (Read or Write) for
% RIO Rack 2 Slot 6
% Fails
% VFD's 05 thru 08 Setpoints %
SOR BST XIC N25:30/12 NXB XIC N25:35/12 BND BST TON T51:60 0.01 200 0 NXB XIC T51:60/DN OTL B3:15/10 BND EOR
%   N25:30/12  MCC5_OE4_BTW_ERROR  "RIO Rack 2 Slot 5 Analog Output Module BTW Error Bit" %
%   N25:35/12  MCC5_OE4_BTR_ERROR  "RIO Rack 2 Slot 5 Analog Output Module BTR Error Bit" %
%   T51:60  ALARM_RK2_SL5_TMR  "Alarm Read or Write Fault RIO Rack 2 Slot 5 TImer" %
%   B3:15/10  ALARM_BT_RK_2_SL_5  "Alarm Block Transfer Read or Write Fault RIO Rack 2 Slot 5" %

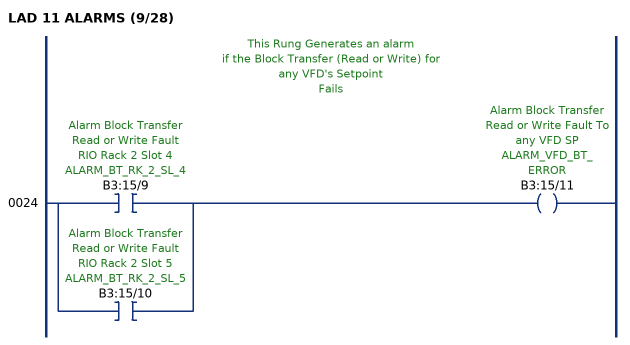
% Rung: 24 %
% This Rung Generates an alarm
% if the Block Transfer (Read or Write) for
% any VFD's Setpoint
% Fails %
SOR BST XIC B3:15/9 NXB XIC B3:15/10 BND OTE B3:15/11 EOR
%   B3:15/9  ALARM_BT_RK_2_SL_4  "Alarm Block Transfer Read or Write Fault RIO Rack 2 Slot 4" %
%   B3:15/10  ALARM_BT_RK_2_SL_5  "Alarm Block Transfer Read or Write Fault RIO Rack 2 Slot 5" %
%   B3:15/11  ALARM_VFD_BT_ERROR  "Alarm Block Transfer Read or Write Fault To any VFD SP" %

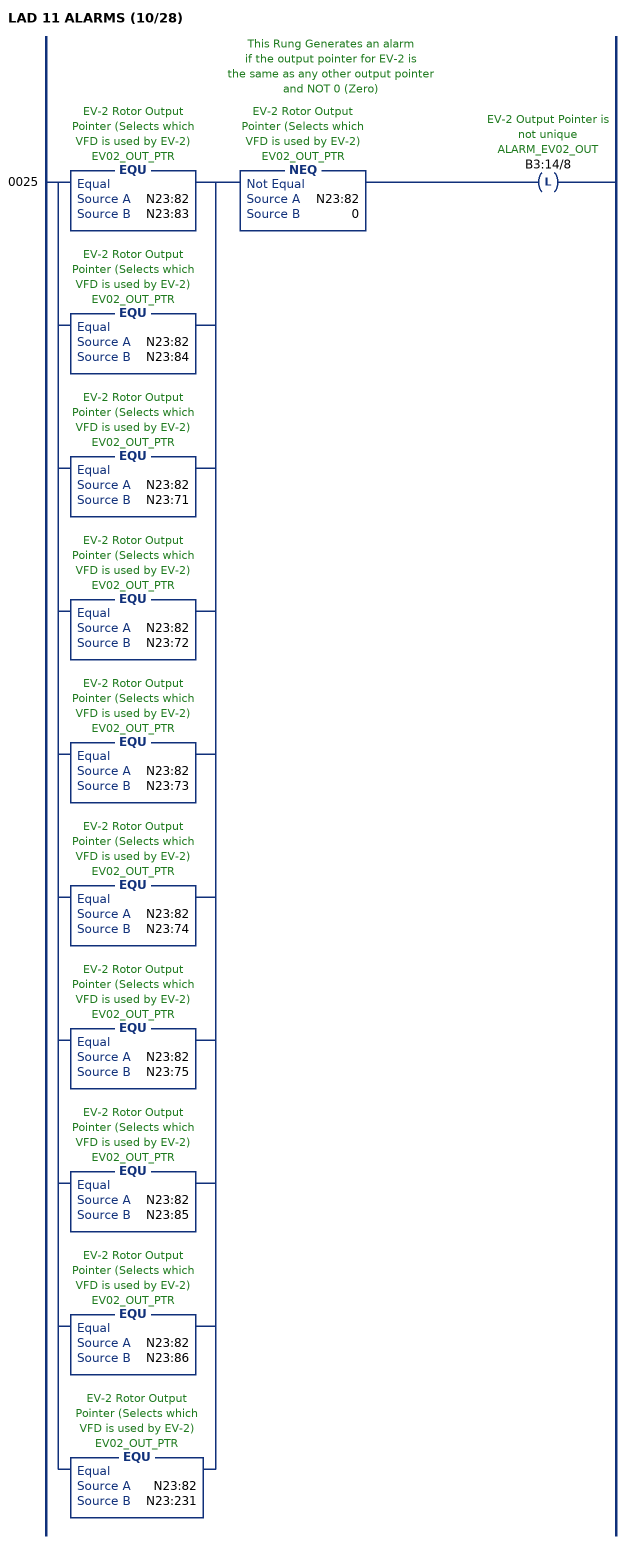
% Rung: 25 %
% This Rung Generates an alarm
% if the output pointer for EV-2 is
% the same as any other output pointer
% and NOT 0 (Zero) %
SOR BST EQU N23:82 N23:83 NXB EQU N23:82 N23:84 NXB EQU N23:82 N23:71 NXB EQU N23:82 N23:72 NXB EQU N23:82 N23:73 NXB EQU N23:82 N23:74 NXB EQU N23:82 N23:75 NXB EQU N23:82 N23:85 NXB EQU N23:82 N23:86 NXB EQU N23:82 N23:231 BND NEQ N23:82 0 OTL B3:14/8 EOR
%   N23:82  EV02_OUT_PTR  "EV-2 Rotor Output Pointer (Selects which VFD is used by EV-2)" %
%   N23:83  EV03_OUT_PTR  "EV-3 Rotor Drive Output Pointer (Selects which VFD is used by EV-3)" %
%   N23:84  AG04_OUT_PTR  "AG-4 Agitator Output Pointer (Selects which VFD is used by AG-4)" %
%   N23:71  FIC211_OUT_PTR  "FIC-21-1 Feed Flow No-1 Output Pointer Determines which VFD is controled by FIC" %
%   N23:72  FIC212_OUT_PTR  "FIC-21-2 Feed Flow No-2 Output Pointer Determines which VFD is controled by FIC" %
%   N23:73  FIC213_OUT_PTR  "FIC-21-3 Feed Flow No-3 Output Pointer Determines which VFD is controled by FIC" %
%   N23:74  FIC214_OUT_PTR  "FIC-21-4 Feed Flow No-4 Output Pointer Determines which VFD is controled by FIC" %
%   N23:75  PIC461_OUT_PTR  "PIC-46-1 Flash Evap Feed Pres Output Pointer Determines which VFD is controled by FIC" %
%   N23:85  EV42_OUT_PTR  "EV-42 Rotor Drive Rotor Output Pointer (Selects which VFD is used by EV-3)" %
%   N23:86  EV20_OUT_PTR  "EV-20 Rotor Drive Rotor Output Pointer (Selects which VFD is used by EV-3)" %
%   N23:231  LIC221_OUT_PTR  "LIC-22-1 Level No-1 Output Pointer Determines which VFD is controled by LIC" %
%   B3:14/8  ALARM_EV02_OUT  "EV-2 Output Pointer is not unique" %

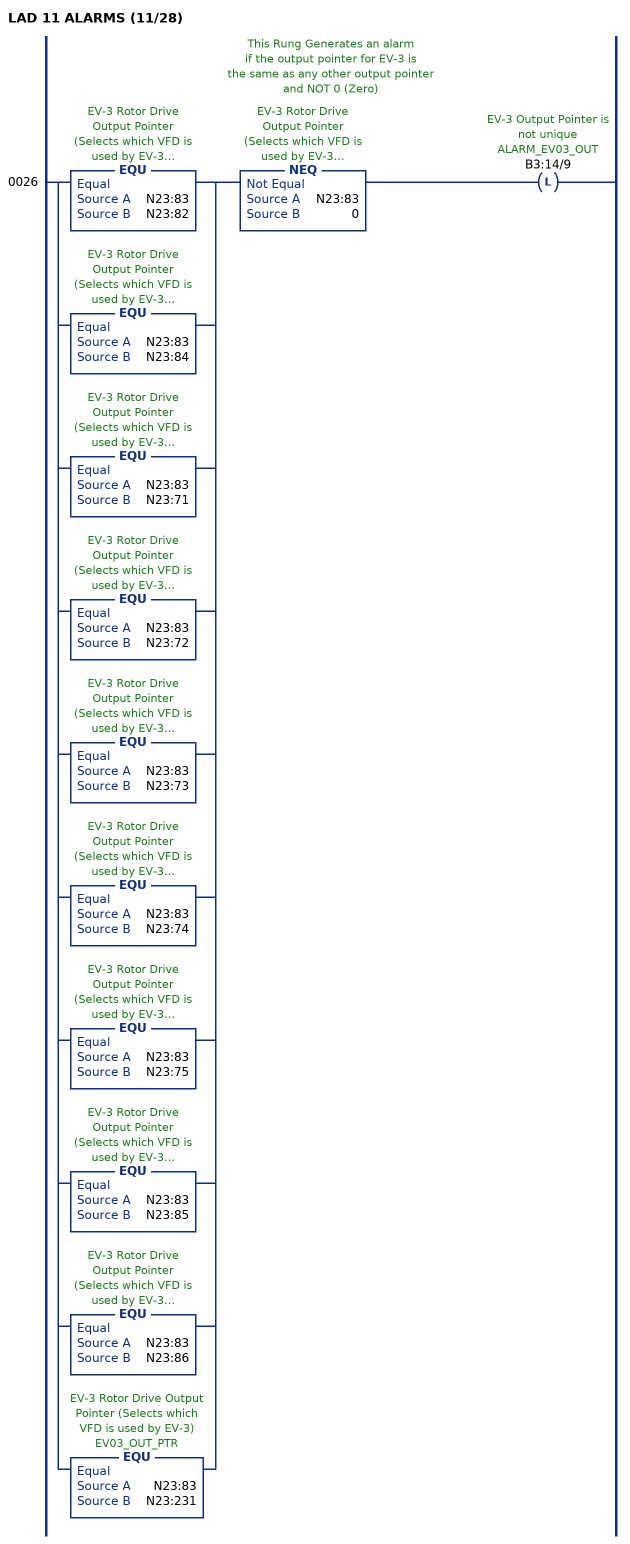
% Rung: 26 %
% This Rung Generates an alarm
% if the output pointer for EV-3 is
% the same as any other output pointer
% and NOT 0 (Zero) %
SOR BST EQU N23:83 N23:82 NXB EQU N23:83 N23:84 NXB EQU N23:83 N23:71 NXB EQU N23:83 N23:72 NXB EQU N23:83 N23:73 NXB EQU N23:83 N23:74 NXB EQU N23:83 N23:75 NXB EQU N23:83 N23:85 NXB EQU N23:83 N23:86 NXB EQU N23:83 N23:231 BND NEQ N23:83 0 OTL B3:14/9 EOR
%   N23:83  EV03_OUT_PTR  "EV-3 Rotor Drive Output Pointer (Selects which VFD is used by EV-3)" %
%   N23:82  EV02_OUT_PTR  "EV-2 Rotor Output Pointer (Selects which VFD is used by EV-2)" %
%   N23:84  AG04_OUT_PTR  "AG-4 Agitator Output Pointer (Selects which VFD is used by AG-4)" %
%   N23:71  FIC211_OUT_PTR  "FIC-21-1 Feed Flow No-1 Output Pointer Determines which VFD is controled by FIC" %
%   N23:72  FIC212_OUT_PTR  "FIC-21-2 Feed Flow No-2 Output Pointer Determines which VFD is controled by FIC" %
%   N23:73  FIC213_OUT_PTR  "FIC-21-3 Feed Flow No-3 Output Pointer Determines which VFD is controled by FIC" %
%   N23:74  FIC214_OUT_PTR  "FIC-21-4 Feed Flow No-4 Output Pointer Determines which VFD is controled by FIC" %
%   N23:75  PIC461_OUT_PTR  "PIC-46-1 Flash Evap Feed Pres Output Pointer Determines which VFD is controled by FIC" %
%   N23:85  EV42_OUT_PTR  "EV-42 Rotor Drive Rotor Output Pointer (Selects which VFD is used by EV-3)" %
%   N23:86  EV20_OUT_PTR  "EV-20 Rotor Drive Rotor Output Pointer (Selects which VFD is used by EV-3)" %
%   N23:231  LIC221_OUT_PTR  "LIC-22-1 Level No-1 Output Pointer Determines which VFD is controled by LIC" %
%   B3:14/9  ALARM_EV03_OUT  "EV-3 Output Pointer is not unique" %

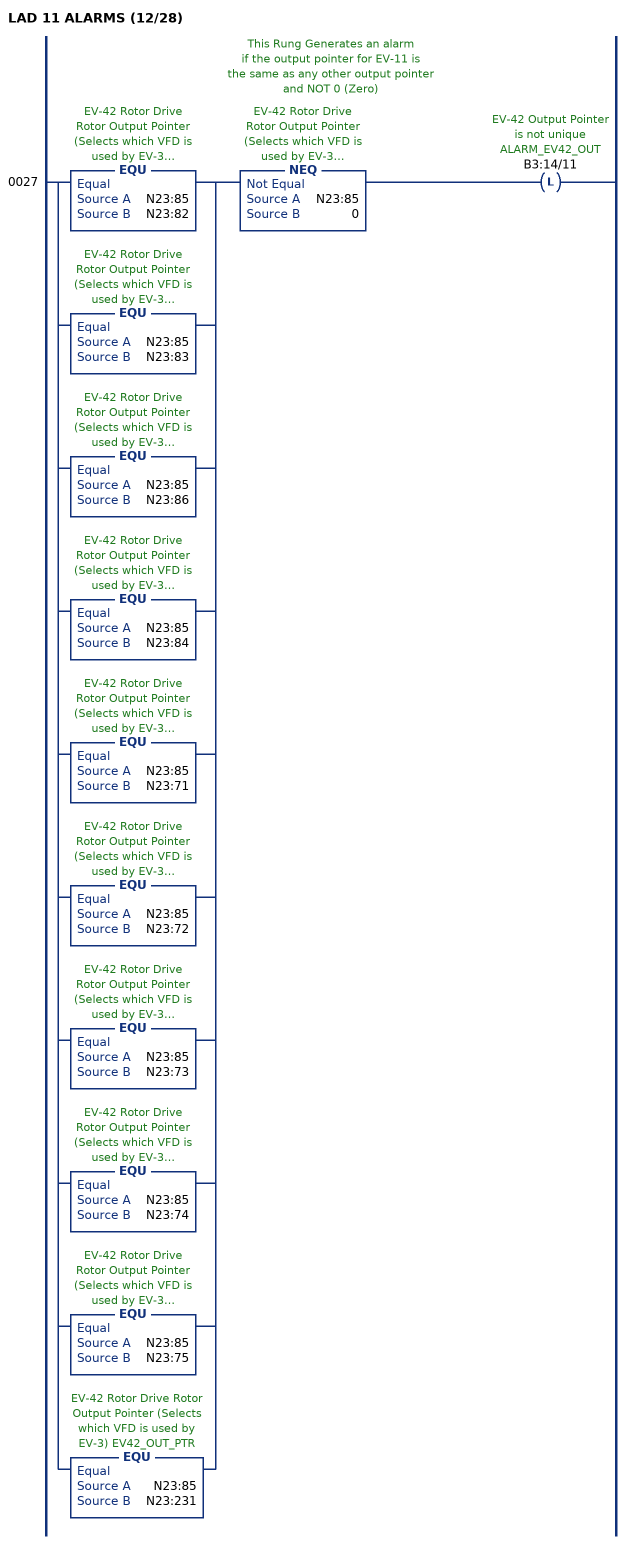
% Rung: 27 %
% This Rung Generates an alarm
% if the output pointer for EV-11 is
% the same as any other output pointer
% and NOT 0 (Zero) %
SOR BST EQU N23:85 N23:82 NXB EQU N23:85 N23:83 NXB EQU N23:85 N23:86 NXB EQU N23:85 N23:84 NXB EQU N23:85 N23:71 NXB EQU N23:85 N23:72 NXB EQU N23:85 N23:73 NXB EQU N23:85 N23:74 NXB EQU N23:85 N23:75 NXB EQU N23:85 N23:231 BND NEQ N23:85 0 OTL B3:14/11 EOR
%   N23:85  EV42_OUT_PTR  "EV-42 Rotor Drive Rotor Output Pointer (Selects which VFD is used by EV-3)" %
%   N23:82  EV02_OUT_PTR  "EV-2 Rotor Output Pointer (Selects which VFD is used by EV-2)" %
%   N23:83  EV03_OUT_PTR  "EV-3 Rotor Drive Output Pointer (Selects which VFD is used by EV-3)" %
%   N23:86  EV20_OUT_PTR  "EV-20 Rotor Drive Rotor Output Pointer (Selects which VFD is used by EV-3)" %
%   N23:84  AG04_OUT_PTR  "AG-4 Agitator Output Pointer (Selects which VFD is used by AG-4)" %
%   N23:71  FIC211_OUT_PTR  "FIC-21-1 Feed Flow No-1 Output Pointer Determines which VFD is controled by FIC" %
%   N23:72  FIC212_OUT_PTR  "FIC-21-2 Feed Flow No-2 Output Pointer Determines which VFD is controled by FIC" %
%   N23:73  FIC213_OUT_PTR  "FIC-21-3 Feed Flow No-3 Output Pointer Determines which VFD is controled by FIC" %
%   N23:74  FIC214_OUT_PTR  "FIC-21-4 Feed Flow No-4 Output Pointer Determines which VFD is controled by FIC" %
%   N23:75  PIC461_OUT_PTR  "PIC-46-1 Flash Evap Feed Pres Output Pointer Determines which VFD is controled by FIC" %
%   N23:231  LIC221_OUT_PTR  "LIC-22-1 Level No-1 Output Pointer Determines which VFD is controled by LIC" %
%   B3:14/11  ALARM_EV42_OUT  "EV-42 Output Pointer is not unique" %

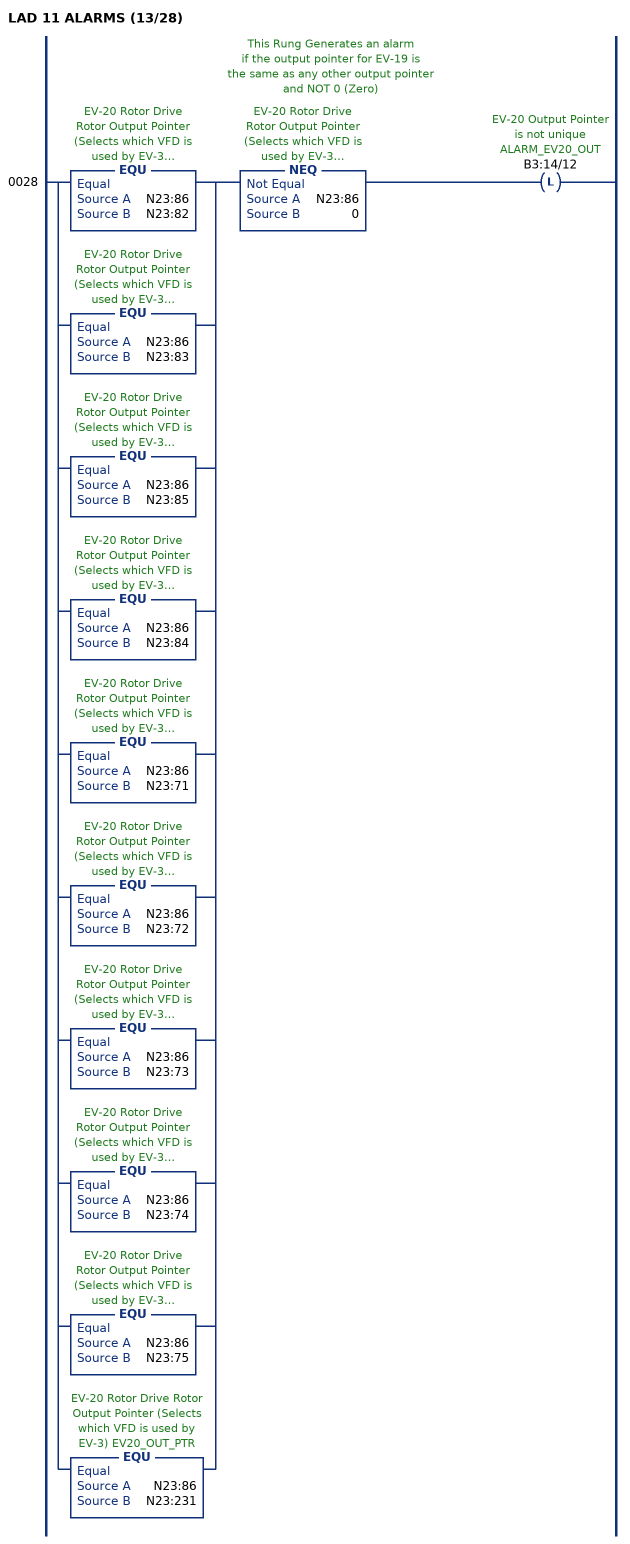
% Rung: 28 %
% This Rung Generates an alarm
% if the output pointer for EV-19 is
% the same as any other output pointer
% and NOT 0 (Zero) %
SOR BST EQU N23:86 N23:82 NXB EQU N23:86 N23:83 NXB EQU N23:86 N23:85 NXB EQU N23:86 N23:84 NXB EQU N23:86 N23:71 NXB EQU N23:86 N23:72 NXB EQU N23:86 N23:73 NXB EQU N23:86 N23:74 NXB EQU N23:86 N23:75 NXB EQU N23:86 N23:231 BND NEQ N23:86 0 OTL B3:14/12 EOR
%   N23:86  EV20_OUT_PTR  "EV-20 Rotor Drive Rotor Output Pointer (Selects which VFD is used by EV-3)" %
%   N23:82  EV02_OUT_PTR  "EV-2 Rotor Output Pointer (Selects which VFD is used by EV-2)" %
%   N23:83  EV03_OUT_PTR  "EV-3 Rotor Drive Output Pointer (Selects which VFD is used by EV-3)" %
%   N23:85  EV42_OUT_PTR  "EV-42 Rotor Drive Rotor Output Pointer (Selects which VFD is used by EV-3)" %
%   N23:84  AG04_OUT_PTR  "AG-4 Agitator Output Pointer (Selects which VFD is used by AG-4)" %
%   N23:71  FIC211_OUT_PTR  "FIC-21-1 Feed Flow No-1 Output Pointer Determines which VFD is controled by FIC" %
%   N23:72  FIC212_OUT_PTR  "FIC-21-2 Feed Flow No-2 Output Pointer Determines which VFD is controled by FIC" %
%   N23:73  FIC213_OUT_PTR  "FIC-21-3 Feed Flow No-3 Output Pointer Determines which VFD is controled by FIC" %
%   N23:74  FIC214_OUT_PTR  "FIC-21-4 Feed Flow No-4 Output Pointer Determines which VFD is controled by FIC" %
%   N23:75  PIC461_OUT_PTR  "PIC-46-1 Flash Evap Feed Pres Output Pointer Determines which VFD is controled by FIC" %
%   N23:231  LIC221_OUT_PTR  "LIC-22-1 Level No-1 Output Pointer Determines which VFD is controled by LIC" %
%   B3:14/12  ALARM_EV20_OUT  "EV-20 Output Pointer is not unique" %

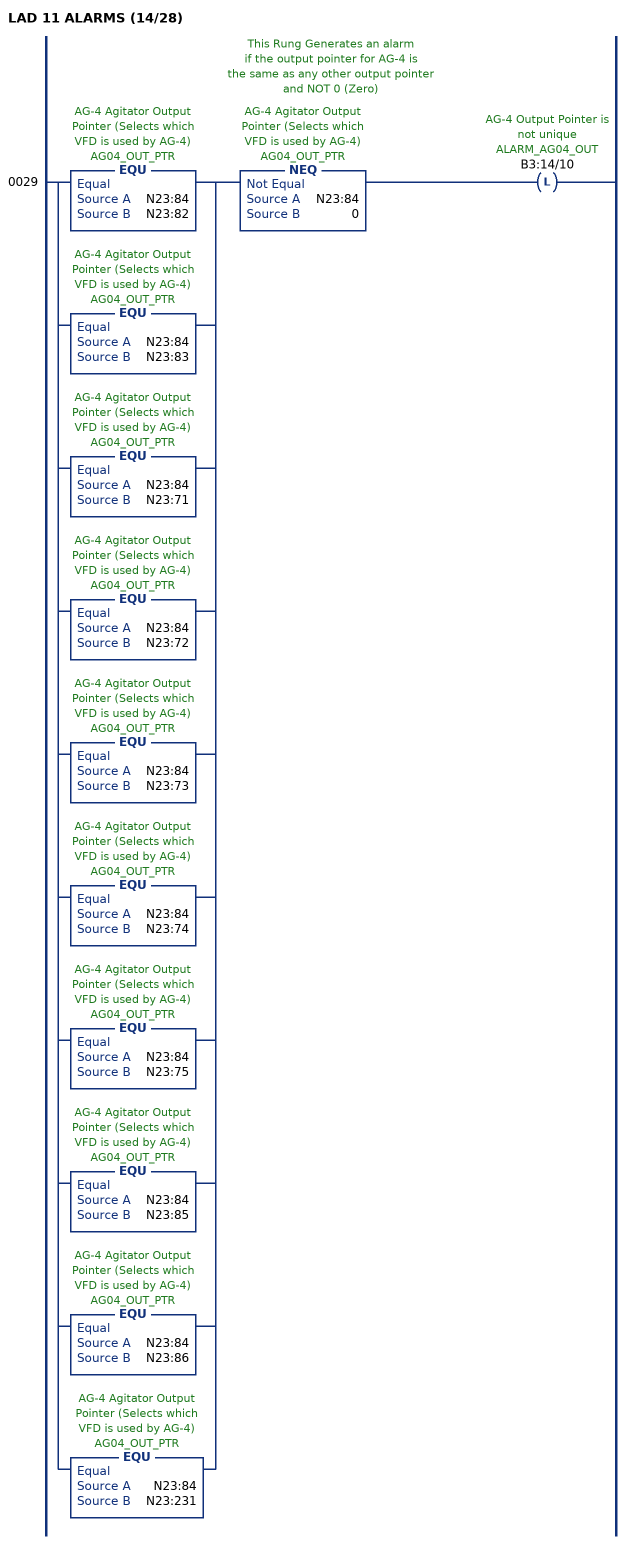
% Rung: 29 %
% This Rung Generates an alarm
% if the output pointer for AG-4 is
% the same as any other output pointer
% and NOT 0 (Zero) %
SOR BST EQU N23:84 N23:82 NXB EQU N23:84 N23:83 NXB EQU N23:84 N23:71 NXB EQU N23:84 N23:72 NXB EQU N23:84 N23:73 NXB EQU N23:84 N23:74 NXB EQU N23:84 N23:75 NXB EQU N23:84 N23:85 NXB EQU N23:84 N23:86 NXB EQU N23:84 N23:231 BND NEQ N23:84 0 OTL B3:14/10 EOR
%   N23:84  AG04_OUT_PTR  "AG-4 Agitator Output Pointer (Selects which VFD is used by AG-4)" %
%   N23:82  EV02_OUT_PTR  "EV-2 Rotor Output Pointer (Selects which VFD is used by EV-2)" %
%   N23:83  EV03_OUT_PTR  "EV-3 Rotor Drive Output Pointer (Selects which VFD is used by EV-3)" %
%   N23:71  FIC211_OUT_PTR  "FIC-21-1 Feed Flow No-1 Output Pointer Determines which VFD is controled by FIC" %
%   N23:72  FIC212_OUT_PTR  "FIC-21-2 Feed Flow No-2 Output Pointer Determines which VFD is controled by FIC" %
%   N23:73  FIC213_OUT_PTR  "FIC-21-3 Feed Flow No-3 Output Pointer Determines which VFD is controled by FIC" %
%   N23:74  FIC214_OUT_PTR  "FIC-21-4 Feed Flow No-4 Output Pointer Determines which VFD is controled by FIC" %
%   N23:75  PIC461_OUT_PTR  "PIC-46-1 Flash Evap Feed Pres Output Pointer Determines which VFD is controled by FIC" %
%   N23:85  EV42_OUT_PTR  "EV-42 Rotor Drive Rotor Output Pointer (Selects which VFD is used by EV-3)" %
%   N23:86  EV20_OUT_PTR  "EV-20 Rotor Drive Rotor Output Pointer (Selects which VFD is used by EV-3)" %
%   N23:231  LIC221_OUT_PTR  "LIC-22-1 Level No-1 Output Pointer Determines which VFD is controled by LIC" %
%   B3:14/10  ALARM_AG04_OUT  "AG-4 Output Pointer is not unique" %

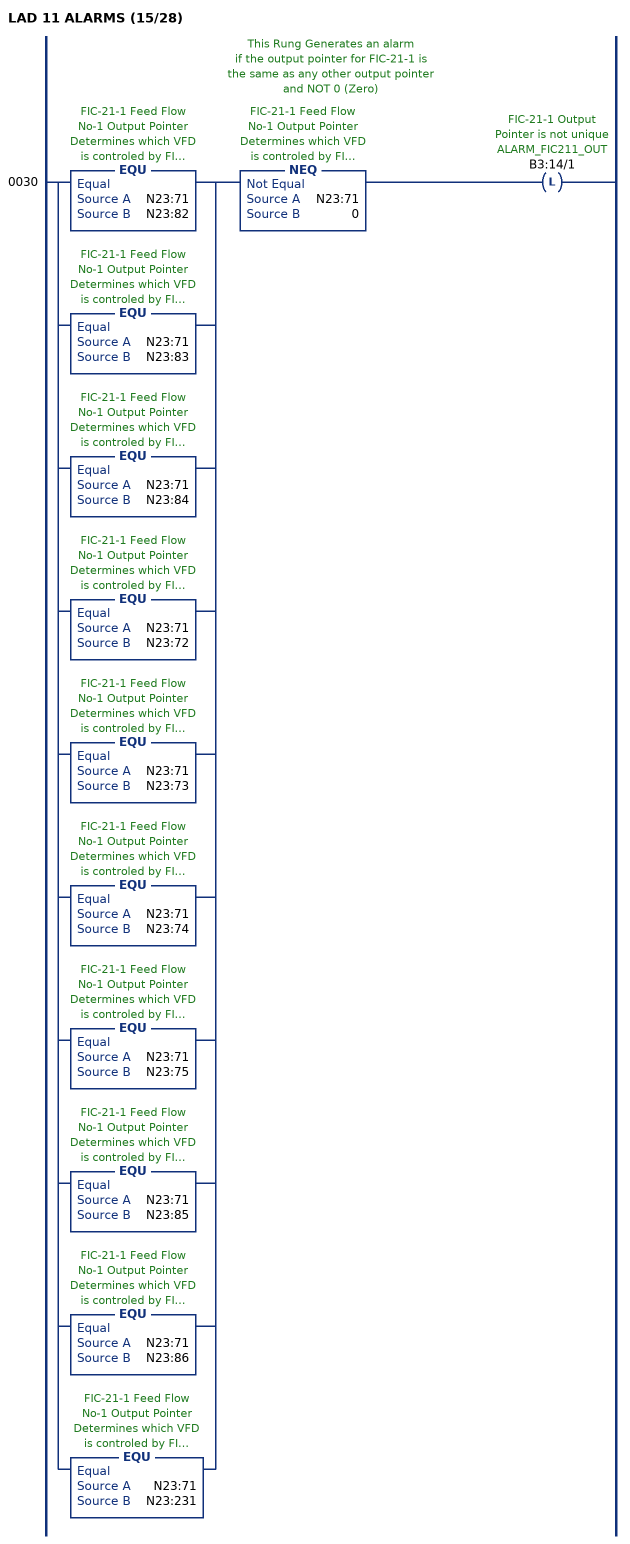
% Rung: 30 %
% This Rung Generates an alarm
% if the output pointer for FIC-21-1 is
% the same as any other output pointer
% and NOT 0 (Zero) %
SOR BST EQU N23:71 N23:82 NXB EQU N23:71 N23:83 NXB EQU N23:71 N23:84 NXB EQU N23:71 N23:72 NXB EQU N23:71 N23:73 NXB EQU N23:71 N23:74 NXB EQU N23:71 N23:75 NXB EQU N23:71 N23:85 NXB EQU N23:71 N23:86 NXB EQU N23:71 N23:231 BND NEQ N23:71 0 OTL B3:14/1 EOR
%   N23:71  FIC211_OUT_PTR  "FIC-21-1 Feed Flow No-1 Output Pointer Determines which VFD is controled by FIC" %
%   N23:82  EV02_OUT_PTR  "EV-2 Rotor Output Pointer (Selects which VFD is used by EV-2)" %
%   N23:83  EV03_OUT_PTR  "EV-3 Rotor Drive Output Pointer (Selects which VFD is used by EV-3)" %
%   N23:84  AG04_OUT_PTR  "AG-4 Agitator Output Pointer (Selects which VFD is used by AG-4)" %
%   N23:72  FIC212_OUT_PTR  "FIC-21-2 Feed Flow No-2 Output Pointer Determines which VFD is controled by FIC" %
%   N23:73  FIC213_OUT_PTR  "FIC-21-3 Feed Flow No-3 Output Pointer Determines which VFD is controled by FIC" %
%   N23:74  FIC214_OUT_PTR  "FIC-21-4 Feed Flow No-4 Output Pointer Determines which VFD is controled by FIC" %
%   N23:75  PIC461_OUT_PTR  "PIC-46-1 Flash Evap Feed Pres Output Pointer Determines which VFD is controled by FIC" %
%   N23:85  EV42_OUT_PTR  "EV-42 Rotor Drive Rotor Output Pointer (Selects which VFD is used by EV-3)" %
%   N23:86  EV20_OUT_PTR  "EV-20 Rotor Drive Rotor Output Pointer (Selects which VFD is used by EV-3)" %
%   N23:231  LIC221_OUT_PTR  "LIC-22-1 Level No-1 Output Pointer Determines which VFD is controled by LIC" %
%   B3:14/1  ALARM_FIC211_OUT  "FIC-21-1 Output Pointer is not unique" %

